FUNCTION TFPackCodePresentToZone : INT
VAR_INPUT
	HandlingPackTable : POINTER TO TFHandlingPackTable;
	WorkAreaZone : POINTER TO TFMachinePalletizer_WorkAreaZone;
	WorkArea : INT;
END_VAR
VAR
	w : INT;
	n : INT;
	i : INT;
	a : INT;
END_VAR

TFPackCodePresentToZone := 0; 

FOR w:=MAXHANDLINGPACK TO 1 BY -1 DO
	IF HandlingPackTable^.Table[w,1].PC > 0 THEN
		FOR n:=1 TO MAXZONE DO
			FOR a:=1 TO MAXAREA DO
				IF WorkAreaZone^.Zone[n].WorkArea[a] = WorkArea THEN
					FOR i:=1 TO MAXFORMINGCODE DO
						(* Verifico se il Pacco presente nel WPP è destinato ad una Zona *)
						IF WorkAreaZone^.Zone[n].Code[i] = HandlingPackTable^.Table[w,1].PC THEN
							TFPackCodePresentToZone := HandlingPackTable^.Table[w,1].PC;
							RETURN;
						END_IF
					END_FOR
				END_IF
			END_FOR
		END_FOR
	END_IF
END_FOR

END_FUNCTION

(* stored: Version 1.1.0.1, ProductVersion 3.1.4024.11
   POU TFPackCodePresentToZone: Id {a0adf196-61b4-44cf-bbef-c418284dfa06}, SpecialFunc None *)
